(*~
    <docu>
        <summary>
            Remote tasks delegates its exectuion to C#.
            When this task is invoked a C# method will be called. To initiliaze <code>RemoteTask</code> with C# method use the <code>Initiliaze method</code>.
            <code>
                    partial void PexConstructor(IVortexObject parent, string readableTail, string symbolTail)
                    {
                        _remoteTaskInstance.InitializeExclusively(Create);
                        //_remoteTaskInstance.Initialize(Create);
                    }

                    private bool Create()
                    {
                        //your code.
                        return true;
                    }
            </code>
        </summary>
        <remarks>Inxton is required for this feature to work</remarks>
    </docu>
~*)
FUNCTION_BLOCK RemoteTask EXTENDS TcoCore.TcoTask
VAR
    {attribute clr [RenderIgnore()]}
    _isInitialized : BOOL;
    {attribute clr [RenderIgnore()]}
    _hasException : BOOL;
    {attribute clr [RenderIgnore()]}
    _startSignature : STRING;
    {attribute clr [RenderIgnore()]}
    _doneSignarure : STRING;
END_VAR

IF Execute() THEN
    IF (_invokeRequest) THEN
        IF (NOT THIS^._isInitialized) THEN
            Messenger.Programming('Remote call not initialized.');
        END_IF;
    END_IF

    IF (THIS^._hasException) THEN
        Messenger.Error('Remote execution produced an exception');
        _startSignature := '';
    END_IF;

    DoneWhen(_startSignature <> '' AND_THEN _startSignature = _doneSignarure);
    ThrowWhen(THIS^._hasException);
END_IF

METHOD PUBLIC FB_init : BOOL
VAR_INPUT
    bInitRetains : BOOL; // if TRUE, the retain variables are initialized (warm start / cold start)
    bInCopyCode : BOOL; // if TRUE, the instance afterwards gets moved into the copy code (online change)
    Parent : ITcoObject;
END_VAR
END_METHOD

METHOD PROTECTED OnStart
_startSignature := LINT_TO_STRING(THIS^.Context.Rtc.TickClock());
_doneSignarure := '';
_hasException := FALSE;
END_METHOD

(*~
    <docu>
        <summary>
            Restores this instance to the Ready state. Can be called explicitly or from within one of the restore mechanisms.
            <para>
                See also <see cref="PlcDocu.TcoCore.TcoTask.AutoRestorable()"/>
            </para>
        </summary>
    </docu>
~*)
METHOD Restore : ITcoRestorable
_startSignature := '';
_doneSignarure := '';
_hasException := FALSE;
Restore := SUPER^.Restore();
END_METHOD

END_FUNCTION_BLOCK

(* stored: Version 1.1.0.1, ProductVersion 3.1.4024.9
   POU RemoteTask: Id {3738faf1-80a5-039e-38b6-48e768300728}, SpecialFunc None
   Method FB_init: Id {dc9a8f58-f99b-0a86-0286-db6e53883867}
   Method OnStart: Id {d70ec8ca-6807-0abf-2f72-d3c79b7f975f}
   Method Restore: Id {b0fbafe3-08ed-012b-384f-b833634311e2} *)
